INTERFACE I_State

METHOD CustomerTakesCoin : BOOL
VAR_INPUT
END_VAR
END_METHOD

METHOD CustomerTakesProduct : BOOL
VAR_INPUT
END_VAR
END_METHOD

PROPERTY Description : STRING
GET
END_GET
END_PROPERTY

METHOD InsertCoin : BOOL
VAR_INPUT
END_VAR
END_METHOD

METHOD PressButton : BOOL
VAR_INPUT
END_VAR
END_METHOD

END_INTERFACE

(* stored: Version 1.1.0.1, ProductVersion 3.1.4022.12
   Itf I_State: Id {67fa25c7-395b-45b1-aa93-be1b802d5c77}
   Method CustomerTakesCoin: Id {47404b5c-ddca-4aea-8031-adf74b4f0917}
   Method CustomerTakesProduct: Id {65e19f78-e189-4597-9305-3d02c005492d}
   Property Description: Id {73c4a00a-9bf7-46a2-bda5-50a460eae680}
   Get Get: Id {6c08231c-fb27-4662-b152-ff2228a53d43}
   Method InsertCoin: Id {e75ade87-9030-41e0-9943-09fb025b9cd3}
   Method PressButton: Id {749b9145-65ee-472b-bf26-c831ed44301e} *)
